//---------------------------------------------------------------------------------------------------------------
//
//  HAUD 2023.03.27
//
//
//  fb_Simulation
//
//    !!! NOT FOR USE IN PRODUCTION !!! --> build something from your mind, this gets messy if you do not
//
//  - grouping of xts stations to sync start process
//  - nFirst to nLast xts stations are checked for starting process simultaneously
//  - basic preparation of station target index in PrepareTarget()
//  - handshake with station control for mover transport through station
//
//---------------------------------------------------------------------------------------------------------------
// This SOFTWARE is provided as an Exemple by THE PROVIDER "as is" and "with all faults." THE PROVIDER makes no 
// representations or warranties of any kind concerning the safety, suitability, lack of viruses, inaccuracies, 
// typographical errors, or other harmful components of this SOFTWARE. There are inherent dangers in the use of 
// any software, and you are solely responsible for determining whether this SOFTWARE is compatible with your 
// equipment and other software installed on your equipment. You are also solely responsible for the protection 
// of your equipment and backup of your data, and THE PROVIDER will not be liable for any damages you may suffer 
// in connection with using, modifying, or distributing this SOFTWARE.
//---------------------------------------------------------------------------------------------------------------
FUNCTION_BLOCK fb_Simulation
VAR
  _nProcessId                 : UINT;

  _sCheck                     : STRING;
  _tonProcess                 : Tc2_Standard.TON;
  _tProcess                   : TIME := T#500MS;

  _AllStationMoverPerMinute   : UDINT;
  _nMoverCountTotal           : UDINT;

  _tonPartsPerMinute          : Tc2_Standard.TON;

  {attribute 'displaymode':='bin'}
  _wEnter                     : DWORD;
  {attribute 'displaymode':='bin'}
  _wStart                     : DWORD;
  {attribute 'displaymode':='bin'}
  _wOut                       : DWORD;
  {attribute 'displaymode':='bin'}
  _wGone                      : DWORD;
  {attribute 'displaymode':='bin'}
  _wEnableProcess             : DWORD; // bits switch on stations

  {attribute 'displaymode':='bin'}
  _TargetMask                 : BYTE;

  _stCtrl                     : POINTER TO ARRAY[1..MAX_STATION]  OF ST_STATION_CTRL;
  _stState                    : POINTER TO ARRAY[1..MAX_STATION]  OF ST_STATION_STATE;

  // controlling bits from properties used on the outside
  _bNext,
  _bMoverEnter,
  _bMoverOut                  : BOOL;

  // who is included in process
  // _nFirst to _nLast MUST be in closed consecutive order
  _nProcessState,
  _nStation,
  _nStationCount,
  _nFirstStation,
  _nLastStation               : UINT;

  _nTarget,
  _nFirstTarget,
  _nLastTarget                : UINT;

  _nPreparedTarget            : ARRAY[1..MAX_MOVER]  OF UINT;

  _nMoverCountStartOld,
  _nMoverCountEnterOld,
  _nMoverCountEnter,
  _nMoverCountStart,
  _nMoverPerMinute,
  _nMoverCount,
  _nMoverCountOld             : ARRAY[1..MAX_STATION]  OF UDINT;

  _rCheckRangeLow,
  _rCheckRangeHigh            : LREAL; // position range the mover has to be in for infeed or sending to happen.

  _MessageLevel               : E_MessageType;
  _stMsg                      : ST_Message;
END_VAR

METHOD Check : BOOL

IF (_nFirstStation < 1) OR
   (_nFirstStation > MAX_STATION)
THEN
  _sCheck                     := '_nFirstStation out of bounds';
  RETURN;
END_IF

IF (_nLastStation < 1) OR
   (_nLastStation > MAX_STATION)
THEN
  _sCheck                     := '_nLastStation out of bounds';
  RETURN;
END_IF

IF (_nFirstTarget < 1) OR
   (_nFirstTarget > MAX_STATION)
THEN
  _sCheck                     := '_nFirstTarget out of bounds';
  RETURN;
END_IF

IF (_nLastTarget < 1) OR
   (_nLastTarget > MAX_STATION)
THEN
  _sCheck                     := '_nLastTarget out of bounds';
  RETURN;
END_IF

IF NOT (_stCtrl  <> 0)
THEN
  _sCheck                     := '_stCtrl: missing pointer';
  RETURN;
END_IF

IF NOT (_stState <> 0)
THEN
  _sCheck                     := '_stState: missing pointer';
  RETURN;
END_IF


_sCheck                       := TO_STRING(E_PROGRESS.PROGRESS_DONE);
Check                         := TRUE;
END_METHOD

PROPERTY CheckRangeHigh : lreal
GET
CheckRangeHigh := _rCheckRangeHigh;
END_GET
SET
_rCheckRangeHigh := CheckRangeHigh;
END_SET
END_PROPERTY

PROPERTY CheckRangeLow : lreal
GET
CheckRangeLow := _rCheckRangeLow;
END_GET
SET
_rCheckRangeLow := CheckRangeLow;
END_SET
END_PROPERTY

METHOD Cycle
VAR_INST
  _interAllStationsCounter    : UDINT;

  _rtrigProcessEnter,
  _rtrigProcessStart,
  _rtrigProcess       : ARRAY[1..MAX_STATION] OF Tc2_Standard.R_TRIG;

  _k                  : UINT;
  _wEnable            : DWORD;
END_VAR
//-----------------------------------------------------------------------------------------------------------------
IF NOT Check() THEN RETURN; END_IF
//-----------------------------------------------------------------------------------------------------------------
_nStationCount                              := _nLastStation - _nFirstStation + 1;
//-----------------------------------------------------------------------------------------------------------------
//-----------------------------------------------------------------------------------------------------------------
IF (_nStationCount < 1)
THEN
  RETURN;
END_IF
//-----------------------------------------------------------------------------------------------------------------
//-----------------------------------------------------------------------------------------------------------------
FOR _nStation := _nLastStation TO _nFirstStation BY(-1) 
DO
  CASE _stState^[_nStation].State
  OF
    //-------------------------------------------------------------------------------------------------------------
    E_STATION_STATE.STATION_DISABLE,
    E_STATION_STATE.STATION_ENABLE, 
    E_STATION_STATE.STATION_DETECT_MOVER:
      _wStart   := _wOut    := _wGone       := 0;
      _wEnter                               := DelBit(_wEnter, (_nStation-_nFirstStation));
      IF (GetBit(_wEnableProcess, (_nStation-_nFirstStation)))
      THEN
        IF (_bMoverEnter)
        THEN
          _stCtrl^[_nStation].Cmd           := E_STATION_CTRL.STATION_ENABLE;
        ELSE
          _stCtrl^[_nStation].Cmd           := E_STATION_CTRL.STATION_DISABLE;
        END_IF
      ELSE
        _stCtrl^[_nStation].Cmd             := E_STATION_CTRL.STATION_DISABLE;
      END_IF


    //-------------------------------------------------------------------------------------------------------------
    E_STATION_STATE.STATION_MOVER_ENTER:
      _wEnter                               := SetBit(_wEnter, (_nStation-_nFirstStation));
      IF _bMoverEnter
      THEN
        _tonProcess(IN                      := FALSE, 
                    PT                      := _tProcess);

        _stCtrl^[_nStation].nTargetStation  := 0;

        IF (_tProcess < T#10MS)
        THEN
          IF (_rCheckRangeHigh > _rCheckRangeLow)
          THEN
            IF (_stState^[_nStation].rMoverModPos > _rCheckRangeLow) AND
               (_stState^[_nStation].rMoverModPos < _rCheckRangeHigh)
            THEN
              _stCtrl^[_nStation].Cmd       := E_STATION_CTRL.STATION_MOVER_SEND;
            END_IF
          ELSE
            IF (_stState^[_nStation].rMoverModPos > _rCheckRangeLow) OR
               (_stState^[_nStation].rMoverModPos < _rCheckRangeHigh)
            THEN
              _stCtrl^[_nStation].Cmd       := E_STATION_CTRL.STATION_MOVER_SEND;
            END_IF
          END_IF
        ELSE
          IF (_rCheckRangeHigh > _rCheckRangeLow)
          THEN
            IF (_stState^[_nStation].rMoverModPos > _rCheckRangeLow) AND
               (_stState^[_nStation].rMoverModPos < _rCheckRangeHigh)
            THEN
              _stCtrl^[_nStation].Cmd       := E_STATION_CTRL.STATION_MOVER_ENTER;
            END_IF
          ELSE
            IF (_stState^[_nStation].rMoverModPos > _rCheckRangeLow) OR
               (_stState^[_nStation].rMoverModPos < _rCheckRangeHigh)
            THEN
              _stCtrl^[_nStation].Cmd       := E_STATION_CTRL.STATION_MOVER_ENTER;
            END_IF
          END_IF
        END_IF
      END_IF

    //-------------------------------------------------------------------------------------------------------------
    E_STATION_STATE.STATION_PROCESS_START:
      _wEnter                               := DelBit(_wEnter, (_nStation-_nFirstStation));
      _wStart                               := SetBit(_wStart, (_nStation-_nFirstStation));
  
      // check if ALL XtsStations have mover in place to work
      IF (_wStart = _wEnableProcess)
      THEN
        _tonProcess(IN                      := TRUE, 
                    PT                      := _tProcess);

        IF _tonProcess.Q
        THEN
          PrepareTargets(FALSE);
          _stCtrl^[_nStation].Cmd           := E_STATION_CTRL.STATION_PROCESS_DONE;
        END_IF
      END_IF

    //-------------------------------------------------------------------------------------------------------------
    E_STATION_STATE.STATION_CHECK_NEST:
      _wEnter                               := SetBit(_wEnter, (_nStation-_nFirstStation));
      _wStart                               := DelBit(_wStart, (_nStation-_nFirstStation));
      _tonProcess(IN                        := FALSE, 
                  PT                        := _tProcess);

      IF (_bNext)
      THEN
        // check if ALL XtsStations have nest to work
        IF (_wEnter = _wEnableProcess)
        THEN
          _stCtrl^[_nStation].Cmd           := E_STATION_CTRL.STATION_MOVER_ENTER;
        END_IF
      END_IF

    //-------------------------------------------------------------------------------------------------------------
    E_STATION_STATE.STATION_MOVER_OUT:
      _wOut                                 := SetBit(_wOut, (_nStation-_nFirstStation));
      _tonProcess(IN                        := FALSE, 
                  PT                        := _tProcess);

      IF _bMoverOut
      THEN
        // nest mask for this mover in target station, sender decides what to work in target
        _stCtrl^[_nStation].nMask           := _TargetMask;

        // check if ALL XtsStations have mover to send
        IF (_wOut = _wEnableProcess)
        THEN
          _nProcessState                    := 10;
        END_IF
      END_IF
  END_CASE
END_FOR
//-----------------------------------------------------------------------------------------------------------------
//-----------------------------------------------------------------------------------------------------------------
CASE _nProcessState
OF
10:
  // ctrl has to decide where to send mover; this depends on YOUR decision
  IF PrepareTargets(TRUE)
  THEN
    PrepareTargets(FALSE);
    _nProcessState                          := 30;
  END_IF
END_CASE
CASE _nProcessState
OF
30:
  FOR _nStation := _nLastStation TO _nFirstStation BY(-1) 
  DO
    IF _bNext
    THEN
      // start outfeed of mover
      _stCtrl^[_nStation].Cmd               := E_STATION_CTRL.STATION_MOVER_OUT;
    END_IF

    CASE _stState^[_nStation].State
    OF
      E_STATION_STATE.STATION_MOVER_GONE:
        _wStart   := _wEnter                := 0;
        // whO is gone?
        _wGone                              := SetBit(_wGone, (_nStation-_nFirstStation));
    END_CASE
  END_FOR
  // check if ALL XtsStations are empty
  IF (_wGone = _wEnableProcess)
  THEN
    _nProcessState                          := 40;
    IF (_MessageLevel > E_MessageType.eMessageVerbose)
    THEN
      _stMsg.eType                          := E_MessageType.eMessageSentient;
      _stMsg.eDevice                        := e_Device.MetricsXts + TO_UINT(_nProcessId);
      _stMsg.eSubdevice                     := e_Subdevice.Process_StationCollector;
      _stMsg.iErrorNumber                   := _nProcessId;
      _stMsg.sText                          := concat('ALL MOVER: ', TO_STRING(E_STATION_STATE.STATION_MOVER_GONE));

      f_MessageSet(_stMsg);
    END_IF
  END_IF
END_CASE
CASE _nProcessState
OF
40:
  _nProcessState                            := 0;
  FOR _nStation := _nLastStation TO _nFirstStation BY(-1) 
  DO
    // let XtsStations jump back to disable
    _stCtrl^[_nStation].Cmd                 := E_STATION_CTRL.STATION_MOVER_GONE;
  END_FOR
END_CASE
//-----------------------------------------------------------------------------------------------------------------
//-----------------------------------------------------------------------------------------------------------------
//-----------------------------------------------------------------------------------------------------------------
// Mover per Minute counter all XtsStations in range
//-----------------------------------------------------------------------------------------------------------------
_nMoverCountTotal                           :=
_AllStationMoverPerMinute                   := 0; 
//-----------------------------------------------------------------------------------------------------------------
// mover counter
//-----------------------------------------------------------------------------------------------------------------
FOR _k := _nLastStation TO _nFirstStation BY(-1)
DO
  //---------------------------------------------------------------------------------------------------------------
  _rtrigProcess[_k](CLK:= ( _stCtrl^[_k].Cmd = E_STATION_CTRL.STATION_MOVER_OUT));
  //---------------------------------------------------------------------------------------------------------------
  IF _rtrigProcess[_k].Q
  THEN
    _nMoverCount[_k]                        := _nMoverCount[_k] + 1;

    IF (_MessageLevel > E_MessageType.eMessageError)
    THEN
      _stMsg.eType                          := E_MessageType.eMessageInfo;
      _stMsg.eDevice                        := e_Device.MetricsXts + TO_UINT(_nProcessId);
      _stMsg.eSubdevice                     := e_Subdevice.Process_StationCollector;
      _stMsg.iErrorNumber                   := _k;
      _stMsg.sText                          := concat('MoverCountStation[ ]: ', TO_STRING(_nMoverCount[_k]));
      _stMsg.sText                          := concat(_stMsg.sText, ': E_STATION_CTRL.');
      _stMsg.sText                          := concat(_stMsg.sText, TO_STRING(_stCtrl^[_k].Cmd));
      f_MessageSet(_stMsg);
    END_IF
  END_IF

  //---------------------------------------------------------------------------------------------------------------
  _rtrigProcessStart[_k](CLK:= ( _stState^[_k].State = E_STATION_STATE.STATION_PROCESS_START));
  //---------------------------------------------------------------------------------------------------------------
  IF _rtrigProcessStart[_k].Q
  THEN
    _nMoverCountStart[_k]                   := _nMoverCountStart[_k] + 1;

    IF (_MessageLevel > E_MessageType.eMessageInfo)
    THEN
      _stMsg.eType                          := E_MessageType.eMessageVerbose;
      _stMsg.eDevice                        := e_Device.MetricsXts + TO_UINT(_nProcessId);
                            
      _stMsg.eSubdevice                     := e_Subdevice.Process_StationCollector;
      _stMsg.iErrorNumber                   := _k;
      _stMsg.sText                          := concat('MoverCountStation[ ]: ', TO_STRING(_nMoverCountEnter[_k]));
      _stMsg.sText                          := concat(_stMsg.sText, ': E_STATION_STATE.');
      _stMsg.sText                          := concat(_stMsg.sText, TO_STRING(_stState^[_k].State));
      f_MessageSet(_stMsg);
    END_IF
  END_IF

  //---------------------------------------------------------------------------------------------------------------
  _rtrigProcessEnter[_k](CLK:= ( _stCtrl^[_k].Cmd = E_STATION_CTRL.STATION_MOVER_ENTER));
  //---------------------------------------------------------------------------------------------------------------
  IF _rtrigProcessEnter[_k].Q
  THEN
    _nMoverCountEnter[_k]                   := _nMoverCountEnter[_k] + 1;

    IF (_MessageLevel > E_MessageType.eMessageVerbose)
    THEN
      _stMsg.eType                          := E_MessageType.eMessageSentient;
      _stMsg.eDevice                        := e_Device.MetricsXts + TO_UINT(_nProcessId);
                            
      _stMsg.eSubdevice                     := e_Subdevice.Process_StationCollector;
      _stMsg.iErrorNumber                   := _k;
      _stMsg.sText                          := concat('MoverCountStation[ ]: ', TO_STRING(_nMoverCountEnter[_k]));
      _stMsg.sText                          := concat(_stMsg.sText, ': E_STATION_CTRL.');
      _stMsg.sText                          := concat(_stMsg.sText, TO_STRING(_stCtrl^[_k].Cmd));
      f_MessageSet(_stMsg);
    END_IF
  END_IF
  //---------------------------------------------------------------------------------------------------------------
  //---------------------------------------------------------------------------------------------------------------
  IF _tonPartsperMinute.Q
  THEN
    // count every XtsStation in range
    _nMoverPerMinute[_k]                    := _nMoverCount[_k] - _nMoverCountOld[_k];
    _nMoverCountOld [_k]                    := _nMoverCount[_k];

    _nMoverCountEnterOld [_k]               := _nMoverCountEnter[_k];
    _nMoverCountStartOld [_k]               := _nMoverCountStart[_k];
  END_IF
  // sum up all XtsStations in range
  _AllStationMoverPerMinute                 := _AllStationMoverPerMinute + _nMoverPerMinute[_k]; 
  _interAllStationsCounter                  := _AllStationMoverPerMinute + _nMoverPerMinute[_k];

  // sum up all mover counts in range
  _nMoverCountTotal                         := _nMoverCountTotal + _nMoverCount[_k];
END_FOR
//-----------------------------------------------------------------------------------------------------------------
//-----------------------------------------------------------------------------------------------------------------
// total mover per minute message for all stations in this process
//-----------------------------------------------------------------------------------------------------------------
//-----------------------------------------------------------------------------------------------------------------
IF _tonPartsperMinute.q
THEN
  _tonPartsperMinute(IN:=FALSE);

  IF (_MessageLevel > E_MessageType.eMessageError)
  THEN
    _stMsg.eType                          := E_MessageType.eMessageBatch;
    _stMsg.eDevice                        := e_Device.MetricsXts + TO_UINT(_nProcessId);
  
    _stMsg.eSubdevice                     := e_Subdevice.Process_StationCollector;
    _stMsg.iErrorNumber                   := _nMoverCountTotal;
    _stMsg.sText                          := concat('MoverCountTotal: ', TO_STRING(_nMoverCountTotal));
    _stMsg.sText                          := concat(_stMsg.sText, ': StationLast: ');
    _stMsg.sText                          := concat(_stMsg.sText, TO_STRING(_nLastStation));
    _stMsg.sText                          := concat(_stMsg.sText, ': StationFirst: ');
    _stMsg.sText                          := concat(_stMsg.sText, TO_STRING(_nFirstStation));
    f_MessageSet(_stMsg);
  END_IF
END_IF
//-----------------------------------------------------------------------------------------------------------------
_tonPartsperMinute(IN:= TRUE,   PT:= T#60S);
//-----------------------------------------------------------------------------------------------------------------
//-----------------------------------------------------------------------------------------------------------------
END_METHOD

METHOD PUBLIC DelBit : DWORD
VAR_INPUT
  inVal   : DWORD;
  bitNo   : DINT;
END_VAR
VAR
  wConst : dWORD := 1;
END_VAR
IF ( inVal AND SHL( wConst,bitNo MOD 32 ) ) > 0 THEN
  DelBit := inVal XOR (SHL( wConst,bitNo MOD 32 ));
ELSE
  DelBit := inVal;
END_IF
END_METHOD

METHOD Disable : BOOL
VAR_INPUT
END_VAR
IF NOT (_nLastStation   > 0) OR
   NOT (_nFirstStation  > 0) OR
   NOT (_nLastStation   < MAX_STATION+1) OR
   NOT (_nFirstStation  < MAX_STATION+1)
THEN
  Disable := FALSE;
ELSE
  FOR _nStation := _nLastStation TO _nFirstStation BY(-1) 
  DO
    _stCtrl^[_nStation].Cmd               := E_STATION_CTRL.STATION_DISABLE;
    _stCtrl^[_nStation].nMask             := 0;
  END_FOR

  memset(ADR(_nMoverCount),    0, SIZEOF(_nMoverCount));
  memset(ADR(_nMoverCountOld), 0, SIZEOF(_nMoverCountOld));
  _nProcessState :=  _nTarget             := 0;
  
  Disable := TRUE;
END_IF
END_METHOD

PROPERTY EnableProcess : dword
GET
EnableProcess := _wEnableProcess;
END_GET
SET
_wEnableProcess := EnableProcess;
END_SET
END_PROPERTY

METHOD PUBLIC GetBit : BOOL
VAR_INPUT
  inVal   : DWORD;
  bitNo   : DINT;
END_VAR
VAR
  wConst : DWORD := 1;
END_VAR
IF ( inVal AND SHL( wConst,DINT_TO_SINT(bitNo) MOD 32 ) ) > 0
THEN
  GetBit := TRUE;
ELSE
  GetBit := FALSE;
END_IF
END_METHOD

METHOD Init : BOOL
VAR_INPUT
END_VAR
IF NOT (_nLastStation   > 0) OR
   NOT (_nFirstStation  > 0) OR
   NOT (_nLastStation   < MAX_STATION+1) OR
   NOT (_nFirstStation  < MAX_STATION+1)
THEN
  Init := FALSE;
ELSE
  FOR _nStation := _nLastStation TO _nFirstStation BY(-1) 
  DO
    _stCtrl^[_nStation].Cmd               := E_STATION_CTRL.STATION_INIT;
    _stCtrl^[_nStation].nMask             := 0;
  END_FOR

  memset(ADR(_nMoverCount),    0, SIZEOF(_nMoverCount));
  memset(ADR(_nMoverCountOld), 0, SIZEOF(_nMoverCountOld));
  _nProcessState :=  _nTarget             := 0;
  
  Init := TRUE;
END_IF
END_METHOD

PROPERTY MessageLevel : e_MessageType
GET
MessageLevel := _MessageLevel;
END_GET
SET
VAR
  _ix : uint;
END_VAR
_MessageLevel := MessageLevel;
END_SET
END_PROPERTY

PROPERTY MoverEnter : bool
GET
MoverEnter := _bMoverEnter;
END_GET
SET
_bMoverEnter := MoverEnter;
END_SET
END_PROPERTY

PROPERTY MoverOut : bool
GET
MoverOut := _bMoverOut;
END_GET
SET
_bMoverOut := MoverOut;
END_SET
END_PROPERTY

METHOD Next : BOOL
VAR_INPUT
  Nxt  : Bool;
END_VAR
_bNext := Nxt;
END_METHOD

METHOD PRIVATE PrepareTargets : BOOL
VAR_INPUT
  Execute         : BOOL;
END_VAR
VAR_INST
  _idxStations    : uint;
  _nt,
  _nstate         : UINT;
END_VAR

IF NOT Check() THEN RETURN; END_IF

IF NOT Execute
THEN
  _nstate                             := 0;
END_IF


CASE _nstate
OF
  0:
    IF Execute
    THEN
      _nstate                         := 10;
    END_IF
END_CASE
CASE _nstate
OF
  10:
    _nstate                           := 20;

    FOR _idxStations := _nLastStation TO _nFirstStation BY(-1) 
    DO
      _nt                               := TO_USINT(_nLastTarget - _nTarget);
      _nTarget                          := _nTarget + 1;
  
      _nPreparedTarget[_stState^[_idxStations].nMoverId]  := _nt;
      _stCtrl^[_idxStations].nTargetStation               := TO_USINT(_nt);
  
      IF (_nLastTarget - _nTarget < _nFirstTarget)
      THEN
        _nTarget                        := 0;
      END_IF
    END_FOR
END_CASE
CASE _nstate
OF
  20:
    PrepareTargets                    := TRUE;
END_CASE
END_METHOD

PROPERTY ProcessId : uint
GET
ProcessId := _nProcessId;
END_GET
SET
_nProcessId := ProcessId;
END_SET
END_PROPERTY

PROPERTY ProcessTime : time
GET
ProcessTime := _tProcess;
END_GET
SET
_tProcess := ProcessTime;
END_SET
END_PROPERTY

METHOD PUBLIC SetBit : DWORD
VAR_INPUT
  inVal   : DWORD;
  bitNo   : DINT;
END_VAR
VAR
  wConst  : dWORD := 1;
END_VAR
SetBit := inVal OR SHL( wConst,bitNo MOD 32 );
END_METHOD

PROPERTY StationCount : uint
GET
StationCount := _nStationCount;
END_GET
END_PROPERTY

PROPERTY StationCtrl : pointer to ARRAY[1..MAX_STATION]  OF ST_STATION_CTRL;
SET
_stCtrl := StationCtrl;
END_SET
END_PROPERTY

PROPERTY StationFirst : uint
GET
StationFirst := _nFirstStation;
END_GET
SET
_nFirstStation := StationFirst;
END_SET
END_PROPERTY

PROPERTY StationLast : uint
GET
StationLast := _nLastStation;
END_GET
SET
_nLastStation := StationLast;
END_SET
END_PROPERTY

PROPERTY StationState : POINTER TO ARRAY[1..MAX_STATION]  OF ST_STATION_STATE
SET
_stState := StationState;
END_SET
END_PROPERTY

PROPERTY TargetFirst : uint
GET
TargetFirst := _nFirstTarget;
END_GET
SET
_nFirstTarget := TargetFirst;
END_SET
END_PROPERTY

PROPERTY TargetLast : uint
GET
TargetLast := _nLastTarget;
END_GET
SET
_nLastTarget := TargetLast;
END_SET
END_PROPERTY

PROPERTY TargetMask : byte
GET
TargetMask := _TargetMask;
END_GET
SET
_TargetMask := TargetMask;
END_SET
END_PROPERTY

END_FUNCTION_BLOCK

(* stored: Version 1.1.0.1
   POU fb_Simulation: Id {95547218-5333-4783-8bca-61fa6e34e4a7}, SpecialFunc None
   Folder properties: Id {51511239-3911-4b28-bb06-815fba17ead1}
   Method Check: Id {694de67a-4e59-4f49-9885-0be4e03bbd74}
   Property CheckRangeHigh: Id {f550ee6d-be72-4b7c-ba7c-ff7b600c7bce}
   Get Get: Id {4ff63a5a-a849-40f3-909d-48416303ff09}
   Set Set: Id {45b309d2-7575-413f-b610-5f1eebdc1271}
   Property CheckRangeLow: Id {e6ae35f3-a074-4cb6-9951-51f04f294138}
   Get Get: Id {b439127d-6a03-4995-9e64-565cc2ddaf1c}
   Set Set: Id {8537a4ad-6964-40cf-888e-6df91fac39d5}
   Method Cycle: Id {5de7d7d1-0b78-4d2d-8797-36a2cf0d91ca}
   Method DelBit: Id {70924835-6ae4-4837-a61a-3abca9ac92bf}
   Method Disable: Id {fc0d75f6-4b8a-411a-bacb-0bd6a1cbfff1}
   Property EnableProcess: Id {846a0124-f641-416f-9a0f-1b1ff2f65344}
   Get Get: Id {8c42be0c-10e8-4a71-bf4d-d8d7a5d1653e}
   Set Set: Id {7023e888-724f-48b4-81be-c8ed1c7f8bc3}
   Method GetBit: Id {698f4cd9-5aaa-4948-8330-4ed006eb5d2f}
   Method Init: Id {3c71f824-fa35-410d-88cb-22888870d811}
   Property MessageLevel: Id {134b8feb-f67a-4abc-b532-4dfcccb0892b}
   Get Get: Id {ab0c12ba-b9b9-45ba-a868-16025ccbb7ef}
   Set Set: Id {3d68a2f7-d905-4ed9-9b7f-54a3c4a4b55f}
   Property MoverEnter: Id {087bf083-ec8b-4a8f-b291-4c74557b6372}
   Get Get: Id {0376b55b-a13f-4460-92e6-2a9ddb0f017e}
   Set Set: Id {3bef2022-3643-4016-98c1-73c73fea5614}
   Property MoverOut: Id {01698e23-f0db-4b7b-ae38-64fc57a4ea28}
   Get Get: Id {47abaaf2-2811-45fc-b22d-6c8720f60fce}
   Set Set: Id {e2ee0318-4b14-4609-bc64-cbd249234ffc}
   Method Next: Id {63330e2b-b58d-4dd4-aed5-6c3f323672bb}
   Method PrepareTargets: Id {8e04e3f7-05a5-4812-a2bb-d904c091374f}
   Property ProcessId: Id {83b59b13-5d68-4056-98ce-eb1251c55487}
   Get Get: Id {6c24ac61-9f69-47bb-9c4f-1b32a54bf528}
   Set Set: Id {7cf4cf10-6758-4db5-8a99-e95d5450b526}
   Property ProcessTime: Id {d00419a7-db49-4dbe-aa31-acf19a0e2936}
   Get Get: Id {24facd13-d414-4bb6-b76f-a98920ebcd7f}
   Set Set: Id {5907403c-deff-43eb-8d84-a0de0d2a810b}
   Method SetBit: Id {50b45556-4117-4424-8e04-99a7a8ddf300}
   Property StationCount: Id {8a13de11-7010-44c9-8b19-d9b9a32e8375}
   Get Get: Id {3c9fdc52-c19f-4bb4-87a0-99c7350298cd}
   Property StationCtrl: Id {83803f5f-0b47-46a4-a4b9-14087bd08bb9}
   Set Set: Id {e041ab97-a1e4-4b5b-94c1-ca0431ae2735}
   Property StationFirst: Id {d2de8915-7e68-49ff-9bfd-5b353bb810d6}
   Get Get: Id {775b91a6-93be-4874-960e-58cded1b0fdd}
   Set Set: Id {a51fb2b3-3a10-450f-9eb4-f748fc120193}
   Property StationLast: Id {6aa1df61-bb0a-4645-bee1-71fc1b46d00e}
   Get Get: Id {78a9fd8c-4da9-4370-82bd-241288a835f9}
   Set Set: Id {3eb09a4d-1314-4412-b5ab-245e72f44c71}
   Property StationState: Id {39250f13-fbf7-4949-a663-b45102b295c9}
   Set Set: Id {2850120b-f15e-4fd9-b319-bb074182ffb6}
   Property TargetFirst: Id {a2f15d8b-f149-40e7-916c-1dafe95c52d5}
   Get Get: Id {7ec9dc90-ee4e-4478-9ad4-71684d4c4a2d}
   Set Set: Id {60b2ef36-3b02-44ff-b248-ff358cc20037}
   Property TargetLast: Id {d00b79d6-9d8c-40db-94ff-7fe185df2798}
   Get Get: Id {850f8308-0c62-4637-8025-a5a20d94bc36}
   Set Set: Id {a906dba5-6def-4e19-9ad1-6f2b02714aac}
   Property TargetMask: Id {0902d040-5eff-4257-824b-14abd6cfd0b9}
   Get Get: Id {da5b9f3d-cc87-4305-ba19-ec27e453c528}
   Set Set: Id {54d71b49-c6db-4ffe-9026-bef618ca8f56} *)
